(* PLC project Generated.project, CODESYS CODESYS V3.5 SP19 Patch 1 *)
(* stored: creationDateTime 2026-08-18T01:35:11.329559, modificationDateTime 2026-08-18T01:35:11.329559 *)

(* ======================================================================= 📤 FB_Output — Adaptateur de sortie physique TOR (inversion NO/NC) ─────────────────────────────────────────────────────────────── 🎯 Rôle : Conditionnement et inversion optionnelle de la commande TOR 🔌 Interface : Interface directe vers carte de sortie physique 📄 Doc métier : DOC/AF/AF_Partie-03_Contrats_Composants_v2.1.md §Câblage ======================================================================= *)
FUNCTION_BLOCK FB_Output
  VAR_INPUT
    Command : BOOL;  (* === COMMANDES ET CONFIGURATION === --> [CMD] Ordre logique issu du FB metier appelant *)
    InvertLogic : BOOL;  (* --> [CFG] TRUE = cablage NC (inversion de la sortie) *)
  END_VAR
  VAR_OUTPUT
    State : BOOL;  (* === SORTIES PHYSIQUES === <-- [ACT] Etat logique physique vers la carte de sortie *)
  END_VAR

            

State := Command XOR InvertLogic;

          
END_FUNCTION_BLOCK
